TYPE ChangeOperatingStateProcessArgs :
STRUCT
	///New operating state (e.g. AUTO, MANUAL)
	state: OperatingStates;
END_STRUCT
END_TYPE

(* stored: Version 1.1.0.1, ProductVersion 3.1.4019.2
   DUT ChangeOperatingStateProcessArgs: Id {13a46553-3118-421f-8633-a8e3e9a302cc} *)
